ABB RobotStudio station: ScanAndPose_20251115-125702.rsstn

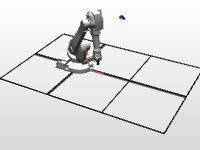
Station ScanAndPose (saved by RobotStudio 6.8.8307.1040)
Controller System1
  mechanical unit ROB_1: IRB1600_10_145__01, 6 joints, base frame (0, 0, 0) mm
Layout (positions relative to the parent item):
  - IRB1600_10_145__01 [mechanism, from Robots\IRB1600_10_145_G_01.rslib] at (0, 0, 0) mm; joint values [-0.4986, 0.5578, 0.834, 0, 0.1791, -0.4986] (rad or m)
Targets, tools, work objects and paths stored in the station, written as RAPID:
! task T_ROB1
MODULE Module1
  CONST robtarget home:=[[806.291651246,0,1154],[0.5,0,0.866025404,0],[0,0,0,0],[9E+09,9E+09,9E+09,9E+09,9E+09,9E+09]];
ENDMODULE

! task T_ROB1
MODULE TesterModule
  PROC testManualMove()
  ENDPROC
ENDMODULE

! task T_ROB1
MODULE MainModule
  PROC main()
    testManualMove;
  ENDPROC
ENDMODULE

